FUNCTION_BLOCK FB_HNHT_CentralMachineHeating EXTENDS FB_SystemContinous
VAR_INPUT
END_VAR
VAR_OUTPUT
END_VAR
VAR
	//default parameters
	localDefaultParameters : ST_HNHT_CentralMachineHeatingDefaultParameters;
	
	//pumps
	stPU300DefaultParameters : ST_PumpGrundfosMagna3DefaultParameters := (tTaskCycleTime := GlobalVariables.tTaskCycleTime_MAIN, tCtrlCycleTime := GlobalVariables.tCtrlCycleTime_MAIN);
	PU300 : FB_PumpGrundfosMagna3 := (ST_DefaultParameters := stPU300DefaultParameters);;

	//valves
	stSV300DefaultParameters : ST_DiscreteValveDefaultParameters := (nFeedback := 0);
	SV300 : FB_DiscreteValve := (ST_DefaultParameters := stSV300DefaultParameters);
	
	//internal variables
	bSetStatusOn_PU300 : BOOL;
	bSetStatusOn_SV300 : BOOL;
	
	bStartTimer : BOOL;
	Timer : TON;
END_VAR

MAIN();
//use timer because valve has no feedback signal (75 sec)
Timer(IN := bStartTimer,
	PT := T#75S);

SV300.GetState_BI();
SV300(bSetStatusOnAutomatic := bSetStatusOn_SV300,
	bAlgorithmPermission := bAlgorithmPermission);
SV300.SetState_BO();

PU300.GetState_Profibus();
PU300(bSetStatusOnAutomatic := bSetStatusOn_PU300,
	bAlgorithmPermission := bAlgorithmPermission,
	fSetPointAutomatic := fSetPoint,
	nControlModeAutomatic := 0);
PU300.SetState_Profibus();

METHOD PROTECTED  CheckError : BOOL
VAR_INPUT
END_VAR
VAR_OUTPUT
	bError : BOOL;
END_VAR
IF PU300.bError THEN
	bError := TRUE;
END_IF
END_METHOD

METHOD PROTECTED  Operational : BOOL
VAR_INPUT
END_VAR
VAR_OUTPUT
	bSwitchToWorking : BOOL := FALSE;
END_VAR
bSetStatusOn_PU300 := TRUE;

IF PU300.bStatusOn THEN
	bSwitchToWorking := TRUE;
END_IF
END_METHOD

METHOD PROTECTED  RampDown : BOOL
VAR_INPUT
END_VAR
VAR_OUTPUT
	bRampDownFinished : BOOL := FALSE;
END_VAR
bSetStatusOn_PU300 := FALSE;

IF NOT PU300.bStatusOn THEN
	bSetStatusOn_SV300 := FALSE;
	bStartTimer := TRUE;
	IF Timer.Q THEN
		bRampDownFinished := TRUE;
		bStartTimer := FALSE;
	END_IF
END_IF
END_METHOD

METHOD PROTECTED  RampUp : BOOL
VAR_INPUT
END_VAR
VAR_OUTPUT
	bRampUpFinished : BOOL := FALSE;
END_VAR
bSetStatusOn_SV300 := TRUE;
bStartTimer := TRUE;

IF Timer.Q THEN
	bRampUpFinished := TRUE;
	bStartTimer := FALSE;
END_IF
END_METHOD

METHOD PROTECTED   SetSetPointLimits : BOOL
VAR_INPUT
END_VAR
aSetPointLimits[1] := localDefaultParameters.aSetPointLimitsRelativeSpeed[1];
aSetPointLimits[2] := localDefaultParameters.aSetPointLimitsRelativeSpeed[2];
END_METHOD

METHOD PROTECTED  SetState : BOOL
VAR_INPUT
END_VAR
VAR_OUTPUT
END_VAR
fOperatingPoint := PU300.fOperatingPoint;

controlState.bStatusOn := bSetStatusOn;
setPointState.aSetPointLimits := aSetPointLimits;
setPointState.fSetPoint := fSetPoint;
setPointState.fOperatingPoint := fOperatingPoint;
setPointState.sSetPointUnit := 'percent';
setPointState.sOperatingPointUnit := 'percent';
END_METHOD

METHOD PROTECTED  Working : BOOL
VAR_INPUT
END_VAR
VAR_OUTPUT
	bSwitchToOperational : BOOL := FALSE;
END_VAR
//empty method
END_METHOD

END_FUNCTION_BLOCK

(* stored: Version 1.1.0.1, ProductVersion 3.1.4024.10
   POU FB_HNHT_CentralMachineHeating: Id {fb1b3375-2b59-4861-bcd1-1213b5b09ae0}, SpecialFunc None
   Method CheckError: Id {c0d9f16c-aba7-43a2-978a-fcedde11b366}
   Method Operational: Id {c847f0bb-451c-4e31-a490-f4280637fbd6}
   Method RampDown: Id {1fdc9863-7f94-466d-95b8-747503f0b82d}
   Method RampUp: Id {ec4d94cd-1da8-44a5-9aaf-95bda85fc2db}
   Method SetSetPointLimits: Id {d9648c5d-1503-4166-94b1-225e1ce0ae2a}
   Method SetState: Id {4e2ea92d-ea0a-4d3f-bc29-d3387dc8f5c1}
   Method Working: Id {e3fbd5c7-b6d4-4929-9e71-72d696dc7a91} *)
